afSi[0  , 0] := 1.00000E+01; afSi[0  , 1] := 6.81245E-01;
afSi[1  , 0] := 1.99800E+01; afSi[1  , 1] := 1.16318E-01;
afSi[2  , 0] := 2.99600E+01; afSi[2  , 1] := 1.82962E-01;
afSi[3  , 0] := 3.99400E+01; afSi[3  , 1] := 2.59571E-01;
afSi[4  , 0] := 4.99200E+01; afSi[4  , 1] := 3.13998E-01;
afSi[5  , 0] := 5.99000E+01; afSi[5  , 1] := 3.46321E-01;
afSi[6  , 0] := 6.98800E+01; afSi[6  , 1] := 3.63846E-01;
afSi[7  , 0] := 7.98600E+01; afSi[7  , 1] := 3.72124E-01;
afSi[8  , 0] := 8.98400E+01; afSi[8  , 1] := 3.76682E-01;
afSi[9  , 0] := 9.98200E+01; afSi[9  , 1] := 7.19156E+00;
afSi[10 , 0] := 1.09800E+02; afSi[10 , 1] := 8.20881E+00;
afSi[11 , 0] := 1.19780E+02; afSi[11 , 1] := 8.98291E+00;
afSi[12 , 0] := 1.29760E+02; afSi[12 , 1] := 9.38953E+00;
afSi[13 , 0] := 1.39740E+02; afSi[13 , 1] := 9.52436E+00;
afSi[14 , 0] := 1.49720E+02; afSi[14 , 1] := 1.01493E+01;
afSi[15 , 0] := 1.59700E+02; afSi[15 , 1] := 1.02033E+01;
afSi[16 , 0] := 1.69680E+02; afSi[16 , 1] := 9.94800E+00;
afSi[17 , 0] := 1.79660E+02; afSi[17 , 1] := 9.62733E+00;
afSi[18 , 0] := 1.89640E+02; afSi[18 , 1] := 9.27233E+00;
afSi[19 , 0] := 1.99620E+02; afSi[19 , 1] := 8.90204E+00;
afSi[20 , 0] := 2.09600E+02; afSi[20 , 1] := 8.52928E+00;
afSi[21 , 0] := 2.19580E+02; afSi[21 , 1] := 8.16149E+00;
afSi[22 , 0] := 2.29560E+02; afSi[22 , 1] := 7.80410E+00;
afSi[23 , 0] := 2.39540E+02; afSi[23 , 1] := 7.46085E+00;
afSi[24 , 0] := 2.49520E+02; afSi[24 , 1] := 7.13329E+00;
afSi[25 , 0] := 2.59500E+02; afSi[25 , 1] := 6.82216E+00;
afSi[26 , 0] := 2.69480E+02; afSi[26 , 1] := 6.52768E+00;
afSi[27 , 0] := 2.79460E+02; afSi[27 , 1] := 6.24948E+00;
afSi[28 , 0] := 2.89440E+02; afSi[28 , 1] := 5.98692E+00;
afSi[29 , 0] := 2.99420E+02; afSi[29 , 1] := 5.73954E+00;
afSi[30 , 0] := 3.09400E+02; afSi[30 , 1] := 5.50624E+00;
afSi[31 , 0] := 3.19380E+02; afSi[31 , 1] := 5.28643E+00;
afSi[32 , 0] := 3.29360E+02; afSi[32 , 1] := 5.07925E+00;
afSi[33 , 0] := 3.39340E+02; afSi[33 , 1] := 4.88381E+00;
afSi[34 , 0] := 3.49320E+02; afSi[34 , 1] := 4.69939E+00;
afSi[35 , 0] := 3.59300E+02; afSi[35 , 1] := 4.52528E+00;
afSi[36 , 0] := 3.69280E+02; afSi[36 , 1] := 4.36069E+00;
afSi[37 , 0] := 3.79260E+02; afSi[37 , 1] := 4.20508E+00;
afSi[38 , 0] := 3.89240E+02; afSi[38 , 1] := 4.05782E+00;
afSi[39 , 0] := 3.99220E+02; afSi[39 , 1] := 3.91835E+00;
afSi[40 , 0] := 4.09200E+02; afSi[40 , 1] := 3.78586E+00;
afSi[41 , 0] := 4.19180E+02; afSi[41 , 1] := 3.65995E+00;
afSi[42 , 0] := 4.29160E+02; afSi[42 , 1] := 3.54031E+00;
afSi[43 , 0] := 4.39140E+02; afSi[43 , 1] := 3.42645E+00;
afSi[44 , 0] := 4.49120E+02; afSi[44 , 1] := 3.31800E+00;
afSi[45 , 0] := 4.59100E+02; afSi[45 , 1] := 3.21480E+00;
afSi[46 , 0] := 4.69080E+02; afSi[46 , 1] := 3.11633E+00;
afSi[47 , 0] := 4.79060E+02; afSi[47 , 1] := 3.02250E+00;
afSi[48 , 0] := 4.89040E+02; afSi[48 , 1] := 2.93291E+00;
afSi[49 , 0] := 4.99020E+02; afSi[49 , 1] := 2.84732E+00;
afSi[50 , 0] := 5.09000E+02; afSi[50 , 1] := 2.76553E+00;
afSi[51 , 0] := 5.18980E+02; afSi[51 , 1] := 2.68738E+00;
afSi[52 , 0] := 5.28960E+02; afSi[52 , 1] := 2.61260E+00;
afSi[53 , 0] := 5.38940E+02; afSi[53 , 1] := 2.54091E+00;
afSi[54 , 0] := 5.48920E+02; afSi[54 , 1] := 2.47233E+00;
afSi[55 , 0] := 5.58900E+02; afSi[55 , 1] := 2.40663E+00;
afSi[56 , 0] := 5.68880E+02; afSi[56 , 1] := 2.34354E+00;
afSi[57 , 0] := 5.78860E+02; afSi[57 , 1] := 2.28303E+00;
afSi[58 , 0] := 5.88840E+02; afSi[58 , 1] := 2.22501E+00;
afSi[59 , 0] := 5.98820E+02; afSi[59 , 1] := 2.16915E+00;
afSi[60 , 0] := 6.08800E+02; afSi[60 , 1] := 2.11548E+00;
afSi[61 , 0] := 6.18780E+02; afSi[61 , 1] := 2.06389E+00;
afSi[62 , 0] := 6.28760E+02; afSi[62 , 1] := 2.01423E+00;
afSi[63 , 0] := 6.38740E+02; afSi[63 , 1] := 1.96636E+00;
afSi[64 , 0] := 6.48720E+02; afSi[64 , 1] := 1.92028E+00;
afSi[65 , 0] := 6.58700E+02; afSi[65 , 1] := 1.87584E+00;
afSi[66 , 0] := 6.68680E+02; afSi[66 , 1] := 1.83301E+00;
afSi[67 , 0] := 6.78660E+02; afSi[67 , 1] := 1.79173E+00;
afSi[68 , 0] := 6.88640E+02; afSi[68 , 1] := 1.75183E+00;
afSi[69 , 0] := 6.98620E+02; afSi[69 , 1] := 1.71334E+00;
afSi[70 , 0] := 7.08600E+02; afSi[70 , 1] := 1.67622E+00;
afSi[71 , 0] := 7.18580E+02; afSi[71 , 1] := 1.64031E+00;
afSi[72 , 0] := 7.28560E+02; afSi[72 , 1] := 1.60563E+00;
afSi[73 , 0] := 7.38540E+02; afSi[73 , 1] := 1.57210E+00;
afSi[74 , 0] := 7.48520E+02; afSi[74 , 1] := 1.53968E+00;
afSi[75 , 0] := 7.58500E+02; afSi[75 , 1] := 1.50829E+00;
afSi[76 , 0] := 7.68480E+02; afSi[76 , 1] := 1.47792E+00;
afSi[77 , 0] := 7.78460E+02; afSi[77 , 1] := 1.44845E+00;
afSi[78 , 0] := 7.88440E+02; afSi[78 , 1] := 1.41998E+00;
afSi[79 , 0] := 7.98420E+02; afSi[79 , 1] := 1.39240E+00;
afSi[80 , 0] := 8.08400E+02; afSi[80 , 1] := 1.36571E+00;
afSi[81 , 0] := 8.18380E+02; afSi[81 , 1] := 1.33980E+00;
afSi[82 , 0] := 8.28360E+02; afSi[82 , 1] := 1.31466E+00;
afSi[83 , 0] := 8.38340E+02; afSi[83 , 1] := 1.29025E+00;
afSi[84 , 0] := 8.48320E+02; afSi[84 , 1] := 1.26656E+00;
afSi[85 , 0] := 8.58300E+02; afSi[85 , 1] := 1.24365E+00;
afSi[86 , 0] := 8.68280E+02; afSi[86 , 1] := 1.22133E+00;
afSi[87 , 0] := 8.78260E+02; afSi[87 , 1] := 1.19966E+00;
afSi[88 , 0] := 8.88240E+02; afSi[88 , 1] := 1.17863E+00;
afSi[89 , 0] := 8.98220E+02; afSi[89 , 1] := 1.15820E+00;
afSi[90 , 0] := 9.08200E+02; afSi[90 , 1] := 1.13838E+00;
afSi[91 , 0] := 9.18180E+02; afSi[91 , 1] := 1.11907E+00;
afSi[92 , 0] := 9.28160E+02; afSi[92 , 1] := 1.10028E+00;
afSi[93 , 0] := 9.38140E+02; afSi[93 , 1] := 1.08204E+00;
afSi[94 , 0] := 9.48120E+02; afSi[94 , 1] := 1.06425E+00;
afSi[95 , 0] := 9.58100E+02; afSi[95 , 1] := 1.04696E+00;
afSi[96 , 0] := 9.68080E+02; afSi[96 , 1] := 1.03008E+00;
afSi[97 , 0] := 9.78060E+02; afSi[97 , 1] := 1.01368E+00;
afSi[98 , 0] := 9.88040E+02; afSi[98 , 1] := 9.97755E-01;
afSi[99 , 0] := 9.98020E+02; afSi[99 , 1] := 9.82162E-01;
afSi[100, 0] := 1.00800E+03; afSi[100, 1] := 9.65278E-01;
afSi[101, 0] := 1.01798E+03; afSi[101, 1] := 9.48403E-01;
afSi[102, 0] := 1.02796E+03; afSi[102, 1] := 9.32011E-01;
afSi[103, 0] := 1.03794E+03; afSi[103, 1] := 9.16062E-01;
afSi[104, 0] := 1.04792E+03; afSi[104, 1] := 9.00554E-01;
afSi[105, 0] := 1.05790E+03; afSi[105, 1] := 8.85466E-01;
afSi[106, 0] := 1.06788E+03; afSi[106, 1] := 8.70790E-01;
afSi[107, 0] := 1.07786E+03; afSi[107, 1] := 8.56506E-01;
afSi[108, 0] := 1.08784E+03; afSi[108, 1] := 8.42603E-01;
afSi[109, 0] := 1.09782E+03; afSi[109, 1] := 8.29061E-01;
afSi[110, 0] := 1.10780E+03; afSi[110, 1] := 8.15865E-01;
afSi[111, 0] := 1.11778E+03; afSi[111, 1] := 8.03013E-01;
afSi[112, 0] := 1.12776E+03; afSi[112, 1] := 7.90489E-01;
afSi[113, 0] := 1.13774E+03; afSi[113, 1] := 7.78275E-01;
afSi[114, 0] := 1.14772E+03; afSi[114, 1] := 7.66367E-01;
afSi[115, 0] := 1.15770E+03; afSi[115, 1] := 7.54761E-01;
afSi[116, 0] := 1.16768E+03; afSi[116, 1] := 7.43435E-01;
afSi[117, 0] := 1.17766E+03; afSi[117, 1] := 7.32388E-01;
afSi[118, 0] := 1.18764E+03; afSi[118, 1] := 7.21604E-01;
afSi[119, 0] := 1.19762E+03; afSi[119, 1] := 7.11077E-01;
afSi[120, 0] := 1.20760E+03; afSi[120, 1] := 7.00801E-01;
afSi[121, 0] := 1.21758E+03; afSi[121, 1] := 6.90760E-01;
afSi[122, 0] := 1.22756E+03; afSi[122, 1] := 6.80959E-01;
afSi[123, 0] := 1.23754E+03; afSi[123, 1] := 6.71384E-01;
afSi[124, 0] := 1.24752E+03; afSi[124, 1] := 6.62024E-01;
afSi[125, 0] := 1.25750E+03; afSi[125, 1] := 6.52877E-01;
afSi[126, 0] := 1.26748E+03; afSi[126, 1] := 6.43939E-01;
afSi[127, 0] := 1.27746E+03; afSi[127, 1] := 6.35196E-01;
afSi[128, 0] := 1.28744E+03; afSi[128, 1] := 6.26651E-01;
afSi[129, 0] := 1.29742E+03; afSi[129, 1] := 6.18294E-01;
afSi[130, 0] := 1.30740E+03; afSi[130, 1] := 6.10118E-01;
afSi[131, 0] := 1.31738E+03; afSi[131, 1] := 6.02115E-01;
afSi[132, 0] := 1.32736E+03; afSi[132, 1] := 5.94283E-01;
afSi[133, 0] := 1.33734E+03; afSi[133, 1] := 5.86618E-01;
afSi[134, 0] := 1.34732E+03; afSi[134, 1] := 5.79115E-01;
afSi[135, 0] := 1.35730E+03; afSi[135, 1] := 5.71772E-01;
afSi[136, 0] := 1.36728E+03; afSi[136, 1] := 5.64968E-01;
afSi[137, 0] := 1.37726E+03; afSi[137, 1] := 5.58124E-01;
afSi[138, 0] := 1.38724E+03; afSi[138, 1] := 5.51234E-01;
afSi[139, 0] := 1.39722E+03; afSi[139, 1] := 5.44489E-01;
afSi[140, 0] := 1.40720E+03; afSi[140, 1] := 5.37874E-01;
afSi[141, 0] := 1.41718E+03; afSi[141, 1] := 5.31392E-01;
afSi[142, 0] := 1.42716E+03; afSi[142, 1] := 5.25043E-01;
afSi[143, 0] := 1.43714E+03; afSi[143, 1] := 5.18819E-01;
afSi[144, 0] := 1.44712E+03; afSi[144, 1] := 5.12719E-01;
afSi[145, 0] := 1.45710E+03; afSi[145, 1] := 5.06739E-01;
afSi[146, 0] := 1.46708E+03; afSi[146, 1] := 5.00878E-01;
afSi[147, 0] := 1.47706E+03; afSi[147, 1] := 4.95126E-01;
afSi[148, 0] := 1.48704E+03; afSi[148, 1] := 4.89482E-01;
afSi[149, 0] := 1.49702E+03; afSi[149, 1] := 4.83950E-01;
afSi[150, 0] := 1.50700E+03; afSi[150, 1] := 4.78523E-01;
afSi[151, 0] := 1.51698E+03; afSi[151, 1] := 4.73196E-01;
afSi[152, 0] := 1.52696E+03; afSi[152, 1] := 4.67971E-01;
afSi[153, 0] := 1.53694E+03; afSi[153, 1] := 4.62844E-01;
afSi[154, 0] := 1.54692E+03; afSi[154, 1] := 4.57811E-01;
afSi[155, 0] := 1.55690E+03; afSi[155, 1] := 4.52871E-01;
afSi[156, 0] := 1.56688E+03; afSi[156, 1] := 4.48024E-01;
afSi[157, 0] := 1.57686E+03; afSi[157, 1] := 4.43265E-01;
afSi[158, 0] := 1.58684E+03; afSi[158, 1] := 4.38596E-01;
afSi[159, 0] := 1.59682E+03; afSi[159, 1] := 4.34013E-01;
afSi[160, 0] := 1.60680E+03; afSi[160, 1] := 4.29517E-01;
afSi[161, 0] := 1.61678E+03; afSi[161, 1] := 4.25105E-01;
afSi[162, 0] := 1.62676E+03; afSi[162, 1] := 4.20771E-01;
afSi[163, 0] := 1.63674E+03; afSi[163, 1] := 4.16519E-01;
afSi[164, 0] := 1.64672E+03; afSi[164, 1] := 4.12348E-01;
afSi[165, 0] := 1.65670E+03; afSi[165, 1] := 4.08254E-01;
afSi[166, 0] := 1.66668E+03; afSi[166, 1] := 4.04241E-01;
afSi[167, 0] := 1.67666E+03; afSi[167, 1] := 4.00302E-01;
afSi[168, 0] := 1.68664E+03; afSi[168, 1] := 3.96446E-01;
afSi[169, 0] := 1.69662E+03; afSi[169, 1] := 3.92678E-01;
afSi[170, 0] := 1.70660E+03; afSi[170, 1] := 3.88985E-01;
afSi[171, 0] := 1.71658E+03; afSi[171, 1] := 3.85390E-01;
afSi[172, 0] := 1.72656E+03; afSi[172, 1] := 3.81869E-01;
afSi[173, 0] := 1.73654E+03; afSi[173, 1] := 3.78464E-01;
afSi[174, 0] := 1.74652E+03; afSi[174, 1] := 3.75164E-01;
afSi[175, 0] := 1.75650E+03; afSi[175, 1] := 3.71977E-01;
afSi[176, 0] := 1.76648E+03; afSi[176, 1] := 3.68994E-01;
afSi[177, 0] := 1.77646E+03; afSi[177, 1] := 3.66114E-01;
afSi[178, 0] := 1.78644E+03; afSi[178, 1] := 3.63726E-01;
afSi[179, 0] := 1.79642E+03; afSi[179, 1] := 3.61633E-01;
afSi[180, 0] := 1.80640E+03; afSi[180, 1] := 3.60725E-01;
afSi[181, 0] := 1.81638E+03; afSi[181, 1] := 3.61625E-01;
afSi[182, 0] := 1.82636E+03; afSi[182, 1] := 3.68918E-01;
afSi[183, 0] := 1.83634E+03; afSi[183, 1] := 4.60263E-01;
afSi[184, 0] := 1.84632E+03; afSi[184, 1] := 4.04826E+00;
afSi[185, 0] := 1.85630E+03; afSi[185, 1] := 4.04956E+00;
afSi[186, 0] := 1.86628E+03; afSi[186, 1] := 4.03746E+00;
afSi[187, 0] := 1.87626E+03; afSi[187, 1] := 4.02159E+00;
afSi[188, 0] := 1.88624E+03; afSi[188, 1] := 4.00531E+00;
afSi[189, 0] := 1.89622E+03; afSi[189, 1] := 3.98804E+00;
afSi[190, 0] := 1.90620E+03; afSi[190, 1] := 3.97090E+00;
afSi[191, 0] := 1.91618E+03; afSi[191, 1] := 3.95361E+00;
afSi[192, 0] := 1.92616E+03; afSi[192, 1] := 3.93518E+00;
afSi[193, 0] := 1.93614E+03; afSi[193, 1] := 3.91177E+00;
afSi[194, 0] := 1.94612E+03; afSi[194, 1] := 3.88771E+00;
afSi[195, 0] := 1.95610E+03; afSi[195, 1] := 3.86151E+00;
afSi[196, 0] := 1.96608E+03; afSi[196, 1] := 3.83528E+00;
afSi[197, 0] := 1.97606E+03; afSi[197, 1] := 3.80869E+00;
afSi[198, 0] := 1.98604E+03; afSi[198, 1] := 3.78211E+00;
afSi[199, 0] := 1.99602E+03; afSi[199, 1] := 3.75528E+00;
afSi[200, 0] := 2.00600E+03; afSi[200, 1] := 3.72847E+00;
afSi[201, 0] := 2.01598E+03; afSi[201, 1] := 3.70146E+00;
afSi[202, 0] := 2.02596E+03; afSi[202, 1] := 3.67455E+00;
afSi[203, 0] := 2.03594E+03; afSi[203, 1] := 3.64755E+00;
afSi[204, 0] := 2.04592E+03; afSi[204, 1] := 3.62067E+00;
afSi[205, 0] := 2.05590E+03; afSi[205, 1] := 3.59369E+00;
afSi[206, 0] := 2.06588E+03; afSi[206, 1] := 3.56688E+00;
afSi[207, 0] := 2.07586E+03; afSi[207, 1] := 3.54005E+00;
afSi[208, 0] := 2.08584E+03; afSi[208, 1] := 3.51346E+00;
afSi[209, 0] := 2.09582E+03; afSi[209, 1] := 3.48686E+00;
afSi[210, 0] := 2.10580E+03; afSi[210, 1] := 3.46054E+00;
afSi[211, 0] := 2.11578E+03; afSi[211, 1] := 3.43418E+00;
afSi[212, 0] := 2.12576E+03; afSi[212, 1] := 3.40813E+00;
afSi[213, 0] := 2.13574E+03; afSi[213, 1] := 3.38209E+00;
afSi[214, 0] := 2.14572E+03; afSi[214, 1] := 3.35637E+00;
afSi[215, 0] := 2.15570E+03; afSi[215, 1] := 3.33075E+00;
afSi[216, 0] := 2.16568E+03; afSi[216, 1] := 3.30542E+00;
afSi[217, 0] := 2.17566E+03; afSi[217, 1] := 3.28023E+00;
afSi[218, 0] := 2.18564E+03; afSi[218, 1] := 3.25529E+00;
afSi[219, 0] := 2.19562E+03; afSi[219, 1] := 3.23054E+00;
afSi[220, 0] := 2.20560E+03; afSi[220, 1] := 3.20602E+00;
afSi[221, 0] := 2.21558E+03; afSi[221, 1] := 3.18174E+00;
afSi[222, 0] := 2.22556E+03; afSi[222, 1] := 3.15767E+00;
afSi[223, 0] := 2.23554E+03; afSi[223, 1] := 3.13387E+00;
afSi[224, 0] := 2.24552E+03; afSi[224, 1] := 3.11029E+00;
afSi[225, 0] := 2.25550E+03; afSi[225, 1] := 3.08699E+00;
afSi[226, 0] := 2.26548E+03; afSi[226, 1] := 3.06393E+00;
afSi[227, 0] := 2.27546E+03; afSi[227, 1] := 3.04114E+00;
afSi[228, 0] := 2.28544E+03; afSi[228, 1] := 3.01857E+00;
afSi[229, 0] := 2.29542E+03; afSi[229, 1] := 2.99625E+00;
afSi[230, 0] := 2.30540E+03; afSi[230, 1] := 2.97429E+00;
afSi[231, 0] := 2.31538E+03; afSi[231, 1] := 2.95276E+00;
afSi[232, 0] := 2.32536E+03; afSi[232, 1] := 2.93145E+00;
afSi[233, 0] := 2.33534E+03; afSi[233, 1] := 2.91014E+00;
afSi[234, 0] := 2.34532E+03; afSi[234, 1] := 2.88908E+00;
afSi[235, 0] := 2.35530E+03; afSi[235, 1] := 2.86831E+00;
afSi[236, 0] := 2.36528E+03; afSi[236, 1] := 2.84780E+00;
afSi[237, 0] := 2.37526E+03; afSi[237, 1] := 2.82758E+00;
afSi[238, 0] := 2.38524E+03; afSi[238, 1] := 2.80769E+00;
afSi[239, 0] := 2.39522E+03; afSi[239, 1] := 2.78804E+00;
afSi[240, 0] := 2.40520E+03; afSi[240, 1] := 2.76923E+00;
afSi[241, 0] := 2.41518E+03; afSi[241, 1] := 2.75063E+00;
afSi[242, 0] := 2.42516E+03; afSi[242, 1] := 2.73228E+00;
afSi[243, 0] := 2.43514E+03; afSi[243, 1] := 2.71415E+00;
afSi[244, 0] := 2.44512E+03; afSi[244, 1] := 2.69621E+00;
afSi[245, 0] := 2.45510E+03; afSi[245, 1] := 2.67847E+00;
afSi[246, 0] := 2.46508E+03; afSi[246, 1] := 2.66091E+00;
afSi[247, 0] := 2.47506E+03; afSi[247, 1] := 2.64357E+00;
afSi[248, 0] := 2.48504E+03; afSi[248, 1] := 2.62642E+00;
afSi[249, 0] := 2.49502E+03; afSi[249, 1] := 2.60947E+00;
afSi[250, 0] := 2.50500E+03; afSi[250, 1] := 2.59273E+00;
afSi[251, 0] := 2.51498E+03; afSi[251, 1] := 2.57616E+00;
afSi[252, 0] := 2.52496E+03; afSi[252, 1] := 2.55981E+00;
afSi[253, 0] := 2.53494E+03; afSi[253, 1] := 2.54364E+00;
afSi[254, 0] := 2.54492E+03; afSi[254, 1] := 2.52764E+00;
afSi[255, 0] := 2.55490E+03; afSi[255, 1] := 2.51181E+00;
afSi[256, 0] := 2.56488E+03; afSi[256, 1] := 2.49615E+00;
afSi[257, 0] := 2.57486E+03; afSi[257, 1] := 2.48063E+00;
afSi[258, 0] := 2.58484E+03; afSi[258, 1] := 2.46527E+00;
afSi[259, 0] := 2.59482E+03; afSi[259, 1] := 2.45007E+00;
afSi[260, 0] := 2.60480E+03; afSi[260, 1] := 2.43508E+00;
afSi[261, 0] := 2.61478E+03; afSi[261, 1] := 2.42024E+00;
afSi[262, 0] := 2.62476E+03; afSi[262, 1] := 2.40554E+00;
afSi[263, 0] := 2.63474E+03; afSi[263, 1] := 2.39098E+00;
afSi[264, 0] := 2.64472E+03; afSi[264, 1] := 2.37657E+00;
afSi[265, 0] := 2.65470E+03; afSi[265, 1] := 2.36233E+00;
afSi[266, 0] := 2.66468E+03; afSi[266, 1] := 2.34824E+00;
afSi[267, 0] := 2.67466E+03; afSi[267, 1] := 2.33428E+00;
afSi[268, 0] := 2.68464E+03; afSi[268, 1] := 2.32046E+00;
afSi[269, 0] := 2.69462E+03; afSi[269, 1] := 2.30677E+00;
afSi[270, 0] := 2.70460E+03; afSi[270, 1] := 2.29321E+00;
afSi[271, 0] := 2.71458E+03; afSi[271, 1] := 2.27979E+00;
afSi[272, 0] := 2.72456E+03; afSi[272, 1] := 2.26650E+00;
afSi[273, 0] := 2.73454E+03; afSi[273, 1] := 2.25334E+00;
afSi[274, 0] := 2.74452E+03; afSi[274, 1] := 2.24031E+00;
afSi[275, 0] := 2.75450E+03; afSi[275, 1] := 2.22740E+00;
afSi[276, 0] := 2.76448E+03; afSi[276, 1] := 2.21459E+00;
afSi[277, 0] := 2.77446E+03; afSi[277, 1] := 2.20189E+00;
afSi[278, 0] := 2.78444E+03; afSi[278, 1] := 2.18931E+00;
afSi[279, 0] := 2.79442E+03; afSi[279, 1] := 2.17684E+00;
afSi[280, 0] := 2.80440E+03; afSi[280, 1] := 2.16448E+00;
afSi[281, 0] := 2.81438E+03; afSi[281, 1] := 2.15222E+00;
afSi[282, 0] := 2.82436E+03; afSi[282, 1] := 2.14007E+00;
afSi[283, 0] := 2.83434E+03; afSi[283, 1] := 2.12803E+00;
afSi[284, 0] := 2.84432E+03; afSi[284, 1] := 2.11606E+00;
afSi[285, 0] := 2.85430E+03; afSi[285, 1] := 2.10418E+00;
afSi[286, 0] := 2.86428E+03; afSi[286, 1] := 2.09242E+00;
afSi[287, 0] := 2.87426E+03; afSi[287, 1] := 2.08079E+00;
afSi[288, 0] := 2.88424E+03; afSi[288, 1] := 2.06926E+00;
afSi[289, 0] := 2.89422E+03; afSi[289, 1] := 2.05783E+00;
afSi[290, 0] := 2.90420E+03; afSi[290, 1] := 2.04650E+00;
afSi[291, 0] := 2.91418E+03; afSi[291, 1] := 2.03527E+00;
afSi[292, 0] := 2.92416E+03; afSi[292, 1] := 2.02413E+00;
afSi[293, 0] := 2.93414E+03; afSi[293, 1] := 2.01310E+00;
afSi[294, 0] := 2.94412E+03; afSi[294, 1] := 2.00215E+00;
afSi[295, 0] := 2.95410E+03; afSi[295, 1] := 1.99131E+00;
afSi[296, 0] := 2.96408E+03; afSi[296, 1] := 1.98056E+00;
afSi[297, 0] := 2.97406E+03; afSi[297, 1] := 1.96990E+00;
afSi[298, 0] := 2.98404E+03; afSi[298, 1] := 1.95926E+00;
afSi[299, 0] := 2.99402E+03; afSi[299, 1] := 1.94855E+00;
afSi[300, 0] := 3.00400E+03; afSi[300, 1] := 1.93793E+00;
afSi[301, 0] := 3.01398E+03; afSi[301, 1] := 1.92730E+00;
afSi[302, 0] := 3.02396E+03; afSi[302, 1] := 1.91653E+00;
afSi[303, 0] := 3.03394E+03; afSi[303, 1] := 1.90585E+00;
afSi[304, 0] := 3.04392E+03; afSi[304, 1] := 1.89527E+00;
afSi[305, 0] := 3.05390E+03; afSi[305, 1] := 1.88476E+00;
afSi[306, 0] := 3.06388E+03; afSi[306, 1] := 1.87435E+00;
afSi[307, 0] := 3.07386E+03; afSi[307, 1] := 1.86404E+00;
afSi[308, 0] := 3.08384E+03; afSi[308, 1] := 1.85383E+00;
afSi[309, 0] := 3.09382E+03; afSi[309, 1] := 1.84371E+00;
afSi[310, 0] := 3.10380E+03; afSi[310, 1] := 1.83367E+00;
afSi[311, 0] := 3.11378E+03; afSi[311, 1] := 1.82372E+00;
afSi[312, 0] := 3.12376E+03; afSi[312, 1] := 1.81385E+00;
afSi[313, 0] := 3.13374E+03; afSi[313, 1] := 1.80407E+00;
afSi[314, 0] := 3.14372E+03; afSi[314, 1] := 1.79437E+00;
afSi[315, 0] := 3.15370E+03; afSi[315, 1] := 1.78475E+00;
afSi[316, 0] := 3.16368E+03; afSi[316, 1] := 1.77521E+00;
afSi[317, 0] := 3.17366E+03; afSi[317, 1] := 1.76575E+00;
afSi[318, 0] := 3.18364E+03; afSi[318, 1] := 1.75637E+00;
afSi[319, 0] := 3.19362E+03; afSi[319, 1] := 1.74707E+00;
afSi[320, 0] := 3.20360E+03; afSi[320, 1] := 1.73785E+00;
afSi[321, 0] := 3.21358E+03; afSi[321, 1] := 1.72870E+00;
afSi[322, 0] := 3.22356E+03; afSi[322, 1] := 1.71964E+00;
afSi[323, 0] := 3.23354E+03; afSi[323, 1] := 1.71064E+00;
afSi[324, 0] := 3.24352E+03; afSi[324, 1] := 1.70173E+00;
afSi[325, 0] := 3.25350E+03; afSi[325, 1] := 1.69289E+00;
afSi[326, 0] := 3.26348E+03; afSi[326, 1] := 1.68412E+00;
afSi[327, 0] := 3.27346E+03; afSi[327, 1] := 1.67543E+00;
afSi[328, 0] := 3.28344E+03; afSi[328, 1] := 1.66681E+00;
afSi[329, 0] := 3.29342E+03; afSi[329, 1] := 1.65826E+00;
afSi[330, 0] := 3.30340E+03; afSi[330, 1] := 1.64979E+00;
afSi[331, 0] := 3.31338E+03; afSi[331, 1] := 1.64139E+00;
afSi[332, 0] := 3.32336E+03; afSi[332, 1] := 1.63306E+00;
afSi[333, 0] := 3.33334E+03; afSi[333, 1] := 1.62477E+00;
afSi[334, 0] := 3.34332E+03; afSi[334, 1] := 1.61655E+00;
afSi[335, 0] := 3.35330E+03; afSi[335, 1] := 1.60840E+00;
afSi[336, 0] := 3.36328E+03; afSi[336, 1] := 1.60032E+00;
afSi[337, 0] := 3.37326E+03; afSi[337, 1] := 1.59231E+00;
afSi[338, 0] := 3.38324E+03; afSi[338, 1] := 1.58436E+00;
afSi[339, 0] := 3.39322E+03; afSi[339, 1] := 1.57647E+00;
afSi[340, 0] := 3.40320E+03; afSi[340, 1] := 1.56864E+00;
afSi[341, 0] := 3.41318E+03; afSi[341, 1] := 1.56086E+00;
afSi[342, 0] := 3.42316E+03; afSi[342, 1] := 1.55315E+00;
afSi[343, 0] := 3.43314E+03; afSi[343, 1] := 1.54551E+00;
afSi[344, 0] := 3.44312E+03; afSi[344, 1] := 1.53793E+00;
afSi[345, 0] := 3.45310E+03; afSi[345, 1] := 1.53041E+00;
afSi[346, 0] := 3.46308E+03; afSi[346, 1] := 1.52295E+00;
afSi[347, 0] := 3.47306E+03; afSi[347, 1] := 1.51554E+00;
afSi[348, 0] := 3.48304E+03; afSi[348, 1] := 1.50818E+00;
afSi[349, 0] := 3.49302E+03; afSi[349, 1] := 1.50089E+00;
afSi[350, 0] := 3.50300E+03; afSi[350, 1] := 1.49366E+00;
afSi[351, 0] := 3.51298E+03; afSi[351, 1] := 1.48649E+00;
afSi[352, 0] := 3.52296E+03; afSi[352, 1] := 1.47938E+00;
afSi[353, 0] := 3.53294E+03; afSi[353, 1] := 1.47232E+00;
afSi[354, 0] := 3.54292E+03; afSi[354, 1] := 1.46528E+00;
afSi[355, 0] := 3.55290E+03; afSi[355, 1] := 1.45830E+00;
afSi[356, 0] := 3.56288E+03; afSi[356, 1] := 1.45137E+00;
afSi[357, 0] := 3.57286E+03; afSi[357, 1] := 1.44451E+00;
afSi[358, 0] := 3.58284E+03; afSi[358, 1] := 1.43770E+00;
afSi[359, 0] := 3.59282E+03; afSi[359, 1] := 1.43095E+00;
afSi[360, 0] := 3.60280E+03; afSi[360, 1] := 1.42425E+00;
afSi[361, 0] := 3.61278E+03; afSi[361, 1] := 1.41760E+00;
afSi[362, 0] := 3.62276E+03; afSi[362, 1] := 1.41099E+00;
afSi[363, 0] := 3.63274E+03; afSi[363, 1] := 1.40444E+00;
afSi[364, 0] := 3.64272E+03; afSi[364, 1] := 1.39793E+00;
afSi[365, 0] := 3.65270E+03; afSi[365, 1] := 1.39148E+00;
afSi[366, 0] := 3.66268E+03; afSi[366, 1] := 1.38507E+00;
afSi[367, 0] := 3.67266E+03; afSi[367, 1] := 1.37870E+00;
afSi[368, 0] := 3.68264E+03; afSi[368, 1] := 1.37200E+00;
afSi[369, 0] := 3.69262E+03; afSi[369, 1] := 1.36529E+00;
afSi[370, 0] := 3.70260E+03; afSi[370, 1] := 1.35864E+00;
afSi[371, 0] := 3.71258E+03; afSi[371, 1] := 1.35202E+00;
afSi[372, 0] := 3.72256E+03; afSi[372, 1] := 1.34540E+00;
afSi[373, 0] := 3.73254E+03; afSi[373, 1] := 1.33883E+00;
afSi[374, 0] := 3.74252E+03; afSi[374, 1] := 1.33231E+00;
afSi[375, 0] := 3.75250E+03; afSi[375, 1] := 1.32585E+00;
afSi[376, 0] := 3.76248E+03; afSi[376, 1] := 1.31944E+00;
afSi[377, 0] := 3.77246E+03; afSi[377, 1] := 1.31308E+00;
afSi[378, 0] := 3.78244E+03; afSi[378, 1] := 1.30677E+00;
afSi[379, 0] := 3.79242E+03; afSi[379, 1] := 1.30050E+00;
afSi[380, 0] := 3.80240E+03; afSi[380, 1] := 1.29427E+00;
afSi[381, 0] := 3.81238E+03; afSi[381, 1] := 1.28809E+00;
afSi[382, 0] := 3.82236E+03; afSi[382, 1] := 1.28195E+00;
afSi[383, 0] := 3.83234E+03; afSi[383, 1] := 1.27586E+00;
afSi[384, 0] := 3.84232E+03; afSi[384, 1] := 1.26980E+00;
afSi[385, 0] := 3.85230E+03; afSi[385, 1] := 1.26380E+00;
afSi[386, 0] := 3.86228E+03; afSi[386, 1] := 1.25784E+00;
afSi[387, 0] := 3.87226E+03; afSi[387, 1] := 1.25194E+00;
afSi[388, 0] := 3.88224E+03; afSi[388, 1] := 1.24608E+00;
afSi[389, 0] := 3.89222E+03; afSi[389, 1] := 1.24027E+00;
afSi[390, 0] := 3.90220E+03; afSi[390, 1] := 1.23449E+00;
afSi[391, 0] := 3.91218E+03; afSi[391, 1] := 1.22873E+00;
afSi[392, 0] := 3.92216E+03; afSi[392, 1] := 1.22302E+00;
afSi[393, 0] := 3.93214E+03; afSi[393, 1] := 1.21734E+00;
afSi[394, 0] := 3.94212E+03; afSi[394, 1] := 1.21172E+00;
afSi[395, 0] := 3.95210E+03; afSi[395, 1] := 1.20615E+00;
afSi[396, 0] := 3.96208E+03; afSi[396, 1] := 1.20062E+00;
afSi[397, 0] := 3.97206E+03; afSi[397, 1] := 1.19513E+00;
afSi[398, 0] := 3.98204E+03; afSi[398, 1] := 1.18967E+00;
afSi[399, 0] := 3.99202E+03; afSi[399, 1] := 1.18423E+00;
afSi[400, 0] := 4.00200E+03; afSi[400, 1] := 1.17884E+00;
afSi[401, 0] := 4.01198E+03; afSi[401, 1] := 1.17348E+00;
afSi[402, 0] := 4.02196E+03; afSi[402, 1] := 1.16816E+00;
afSi[403, 0] := 4.03194E+03; afSi[403, 1] := 1.16291E+00;
afSi[404, 0] := 4.04192E+03; afSi[404, 1] := 1.15769E+00;
afSi[405, 0] := 4.05190E+03; afSi[405, 1] := 1.15250E+00;
afSi[406, 0] := 4.06188E+03; afSi[406, 1] := 1.14735E+00;
afSi[407, 0] := 4.07186E+03; afSi[407, 1] := 1.14222E+00;
afSi[408, 0] := 4.08184E+03; afSi[408, 1] := 1.13712E+00;
afSi[409, 0] := 4.09182E+03; afSi[409, 1] := 1.13206E+00;
afSi[410, 0] := 4.10180E+03; afSi[410, 1] := 1.12703E+00;
afSi[411, 0] := 4.11178E+03; afSi[411, 1] := 1.12205E+00;
afSi[412, 0] := 4.12176E+03; afSi[412, 1] := 1.11710E+00;
afSi[413, 0] := 4.13174E+03; afSi[413, 1] := 1.11218E+00;
afSi[414, 0] := 4.14172E+03; afSi[414, 1] := 1.10730E+00;
afSi[415, 0] := 4.15170E+03; afSi[415, 1] := 1.10246E+00;
afSi[416, 0] := 4.16168E+03; afSi[416, 1] := 1.09765E+00;
afSi[417, 0] := 4.17166E+03; afSi[417, 1] := 1.09287E+00;
afSi[418, 0] := 4.18164E+03; afSi[418, 1] := 1.08812E+00;
afSi[419, 0] := 4.19162E+03; afSi[419, 1] := 1.08340E+00;
afSi[420, 0] := 4.20160E+03; afSi[420, 1] := 1.07870E+00;
afSi[421, 0] := 4.21158E+03; afSi[421, 1] := 1.07404E+00;
afSi[422, 0] := 4.22156E+03; afSi[422, 1] := 1.06940E+00;
afSi[423, 0] := 4.23154E+03; afSi[423, 1] := 1.06481E+00;
afSi[424, 0] := 4.24152E+03; afSi[424, 1] := 1.06025E+00;
afSi[425, 0] := 4.25150E+03; afSi[425, 1] := 1.05572E+00;
afSi[426, 0] := 4.26148E+03; afSi[426, 1] := 1.05122E+00;
afSi[427, 0] := 4.27146E+03; afSi[427, 1] := 1.04674E+00;
afSi[428, 0] := 4.28144E+03; afSi[428, 1] := 1.04229E+00;
afSi[429, 0] := 4.29142E+03; afSi[429, 1] := 1.03787E+00;
afSi[430, 0] := 4.30140E+03; afSi[430, 1] := 1.03347E+00;
afSi[431, 0] := 4.31138E+03; afSi[431, 1] := 1.02911E+00;
afSi[432, 0] := 4.32136E+03; afSi[432, 1] := 1.02479E+00;
afSi[433, 0] := 4.33134E+03; afSi[433, 1] := 1.02050E+00;
afSi[434, 0] := 4.34132E+03; afSi[434, 1] := 1.01623E+00;
afSi[435, 0] := 4.35130E+03; afSi[435, 1] := 1.01199E+00;
afSi[436, 0] := 4.36128E+03; afSi[436, 1] := 1.00776E+00;
afSi[437, 0] := 4.37126E+03; afSi[437, 1] := 1.00356E+00;
afSi[438, 0] := 4.38124E+03; afSi[438, 1] := 9.99379E-01;
afSi[439, 0] := 4.39122E+03; afSi[439, 1] := 9.95230E-01;
afSi[440, 0] := 4.40120E+03; afSi[440, 1] := 9.91115E-01;
afSi[441, 0] := 4.41118E+03; afSi[441, 1] := 9.87029E-01;
afSi[442, 0] := 4.42116E+03; afSi[442, 1] := 9.82970E-01;
afSi[443, 0] := 4.43114E+03; afSi[443, 1] := 9.78937E-01;
afSi[444, 0] := 4.44112E+03; afSi[444, 1] := 9.74929E-01;
afSi[445, 0] := 4.45110E+03; afSi[445, 1] := 9.70947E-01;
afSi[446, 0] := 4.46108E+03; afSi[446, 1] := 9.66989E-01;
afSi[447, 0] := 4.47106E+03; afSi[447, 1] := 9.63057E-01;
afSi[448, 0] := 4.48104E+03; afSi[448, 1] := 9.59149E-01;
afSi[449, 0] := 4.49102E+03; afSi[449, 1] := 9.55265E-01;
afSi[450, 0] := 4.50100E+03; afSi[450, 1] := 9.51404E-01;
afSi[451, 0] := 4.51098E+03; afSi[451, 1] := 9.47568E-01;
afSi[452, 0] := 4.52096E+03; afSi[452, 1] := 9.43756E-01;
afSi[453, 0] := 4.53094E+03; afSi[453, 1] := 9.39968E-01;
afSi[454, 0] := 4.54092E+03; afSi[454, 1] := 9.36205E-01;
afSi[455, 0] := 4.55090E+03; afSi[455, 1] := 9.32465E-01;
afSi[456, 0] := 4.56088E+03; afSi[456, 1] := 9.28749E-01;
afSi[457, 0] := 4.57086E+03; afSi[457, 1] := 9.25055E-01;
afSi[458, 0] := 4.58084E+03; afSi[458, 1] := 9.21383E-01;
afSi[459, 0] := 4.59082E+03; afSi[459, 1] := 9.17734E-01;
afSi[460, 0] := 4.60080E+03; afSi[460, 1] := 9.14107E-01;
afSi[461, 0] := 4.61078E+03; afSi[461, 1] := 9.10502E-01;
afSi[462, 0] := 4.62076E+03; afSi[462, 1] := 9.06919E-01;
afSi[463, 0] := 4.63074E+03; afSi[463, 1] := 9.03358E-01;
afSi[464, 0] := 4.64072E+03; afSi[464, 1] := 8.99819E-01;
afSi[465, 0] := 4.65070E+03; afSi[465, 1] := 8.96301E-01;
afSi[466, 0] := 4.66068E+03; afSi[466, 1] := 8.92804E-01;
afSi[467, 0] := 4.67066E+03; afSi[467, 1] := 8.89329E-01;
afSi[468, 0] := 4.68064E+03; afSi[468, 1] := 8.85876E-01;
afSi[469, 0] := 4.69062E+03; afSi[469, 1] := 8.82444E-01;
afSi[470, 0] := 4.70060E+03; afSi[470, 1] := 8.79032E-01;
afSi[471, 0] := 4.71058E+03; afSi[471, 1] := 8.75640E-01;
afSi[472, 0] := 4.72056E+03; afSi[472, 1] := 8.72267E-01;
afSi[473, 0] := 4.73054E+03; afSi[473, 1] := 8.68914E-01;
afSi[474, 0] := 4.74052E+03; afSi[474, 1] := 8.65581E-01;
afSi[475, 0] := 4.75050E+03; afSi[475, 1] := 8.62268E-01;
afSi[476, 0] := 4.76048E+03; afSi[476, 1] := 8.58974E-01;
afSi[477, 0] := 4.77046E+03; afSi[477, 1] := 8.55702E-01;
afSi[478, 0] := 4.78044E+03; afSi[478, 1] := 8.52448E-01;
afSi[479, 0] := 4.79042E+03; afSi[479, 1] := 8.49214E-01;
afSi[480, 0] := 4.80040E+03; afSi[480, 1] := 8.45998E-01;
afSi[481, 0] := 4.81038E+03; afSi[481, 1] := 8.42802E-01;
afSi[482, 0] := 4.82036E+03; afSi[482, 1] := 8.39624E-01;
afSi[483, 0] := 4.83034E+03; afSi[483, 1] := 8.36465E-01;
afSi[484, 0] := 4.84032E+03; afSi[484, 1] := 8.33325E-01;
afSi[485, 0] := 4.85030E+03; afSi[485, 1] := 8.30202E-01;
afSi[486, 0] := 4.86028E+03; afSi[486, 1] := 8.27098E-01;
afSi[487, 0] := 4.87026E+03; afSi[487, 1] := 8.24011E-01;
afSi[488, 0] := 4.88024E+03; afSi[488, 1] := 8.20942E-01;
afSi[489, 0] := 4.89022E+03; afSi[489, 1] := 8.17890E-01;
afSi[490, 0] := 4.90020E+03; afSi[490, 1] := 8.14857E-01;
afSi[491, 0] := 4.91018E+03; afSi[491, 1] := 8.11840E-01;
afSi[492, 0] := 4.92016E+03; afSi[492, 1] := 8.08842E-01;
afSi[493, 0] := 4.93014E+03; afSi[493, 1] := 8.05860E-01;
afSi[494, 0] := 4.94012E+03; afSi[494, 1] := 8.02895E-01;
afSi[495, 0] := 4.95010E+03; afSi[495, 1] := 7.99947E-01;
afSi[496, 0] := 4.96008E+03; afSi[496, 1] := 7.97017E-01;
afSi[497, 0] := 4.97006E+03; afSi[497, 1] := 7.94104E-01;
afSi[498, 0] := 4.98004E+03; afSi[498, 1] := 7.91208E-01;
afSi[499, 0] := 4.99002E+03; afSi[499, 1] := 7.88327E-01;
afSi[500, 0] := 5.00000E+03; afSi[500, 1] := 7.85463E-01;
afSi[501, 0] := 5.05000E+03; afSi[501, 1] := 7.71346E-01;
afSi[502, 0] := 5.10000E+03; afSi[502, 1] := 7.57615E-01;
afSi[503, 0] := 5.15000E+03; afSi[503, 1] := 7.44268E-01;
afSi[504, 0] := 5.20000E+03; afSi[504, 1] := 7.31279E-01;
afSi[505, 0] := 5.25000E+03; afSi[505, 1] := 7.18637E-01;
afSi[506, 0] := 5.30000E+03; afSi[506, 1] := 7.06325E-01;
afSi[507, 0] := 5.35000E+03; afSi[507, 1] := 6.94343E-01;
afSi[508, 0] := 5.40000E+03; afSi[508, 1] := 6.82669E-01;
afSi[509, 0] := 5.45000E+03; afSi[509, 1] := 6.71298E-01;
afSi[510, 0] := 5.50000E+03; afSi[510, 1] := 6.60221E-01;
afSi[511, 0] := 5.55000E+03; afSi[511, 1] := 6.49422E-01;
afSi[512, 0] := 5.60000E+03; afSi[512, 1] := 6.38895E-01;
afSi[513, 0] := 5.65000E+03; afSi[513, 1] := 6.28633E-01;
afSi[514, 0] := 5.70000E+03; afSi[514, 1] := 6.18619E-01;
afSi[515, 0] := 5.75000E+03; afSi[515, 1] := 6.08855E-01;
afSi[516, 0] := 5.80000E+03; afSi[516, 1] := 5.99328E-01;
afSi[517, 0] := 5.85000E+03; afSi[517, 1] := 5.90032E-01;
afSi[518, 0] := 5.90000E+03; afSi[518, 1] := 5.80957E-01;
afSi[519, 0] := 5.95000E+03; afSi[519, 1] := 5.72095E-01;
afSi[520, 0] := 6.00000E+03; afSi[520, 1] := 5.63442E-01;
afSi[521, 0] := 6.05000E+03; afSi[521, 1] := 5.54992E-01;
afSi[522, 0] := 6.10000E+03; afSi[522, 1] := 5.46736E-01;
afSi[523, 0] := 6.15000E+03; afSi[523, 1] := 5.38668E-01;
afSi[524, 0] := 6.20000E+03; afSi[524, 1] := 5.30779E-01;
afSi[525, 0] := 6.25000E+03; afSi[525, 1] := 5.23070E-01;
afSi[526, 0] := 6.30000E+03; afSi[526, 1] := 5.15535E-01;
afSi[527, 0] := 6.35000E+03; afSi[527, 1] := 5.08167E-01;
afSi[528, 0] := 6.40000E+03; afSi[528, 1] := 5.00964E-01;
afSi[529, 0] := 6.45000E+03; afSi[529, 1] := 4.93915E-01;
afSi[530, 0] := 6.50000E+03; afSi[530, 1] := 4.87022E-01;
afSi[531, 0] := 6.55000E+03; afSi[531, 1] := 4.80279E-01;
afSi[532, 0] := 6.60000E+03; afSi[532, 1] := 4.73675E-01;
afSi[533, 0] := 6.65000E+03; afSi[533, 1] := 4.67207E-01;
afSi[534, 0] := 6.70000E+03; afSi[534, 1] := 4.60877E-01;
afSi[535, 0] := 6.75000E+03; afSi[535, 1] := 4.54682E-01;
afSi[536, 0] := 6.80000E+03; afSi[536, 1] := 4.48615E-01;
afSi[537, 0] := 6.85000E+03; afSi[537, 1] := 4.42675E-01;
afSi[538, 0] := 6.90000E+03; afSi[538, 1] := 4.36855E-01;
afSi[539, 0] := 6.95000E+03; afSi[539, 1] := 4.31151E-01;
afSi[540, 0] := 7.00000E+03; afSi[540, 1] := 4.25560E-01;
afSi[541, 0] := 7.05000E+03; afSi[541, 1] := 4.20081E-01;
afSi[542, 0] := 7.10000E+03; afSi[542, 1] := 4.14712E-01;
afSi[543, 0] := 7.15000E+03; afSi[543, 1] := 4.09450E-01;
afSi[544, 0] := 7.20000E+03; afSi[544, 1] := 4.04294E-01;
afSi[545, 0] := 7.25000E+03; afSi[545, 1] := 3.99235E-01;
afSi[546, 0] := 7.30000E+03; afSi[546, 1] := 3.94270E-01;
afSi[547, 0] := 7.35000E+03; afSi[547, 1] := 3.89406E-01;
afSi[548, 0] := 7.40000E+03; afSi[548, 1] := 3.84633E-01;
afSi[549, 0] := 7.45000E+03; afSi[549, 1] := 3.79947E-01;
afSi[550, 0] := 7.50000E+03; afSi[550, 1] := 3.75353E-01;
afSi[551, 0] := 7.55000E+03; afSi[551, 1] := 3.70843E-01;
afSi[552, 0] := 7.60000E+03; afSi[552, 1] := 3.66417E-01;
afSi[553, 0] := 7.65000E+03; afSi[553, 1] := 3.62071E-01;
afSi[554, 0] := 7.70000E+03; afSi[554, 1] := 3.57805E-01;
afSi[555, 0] := 7.75000E+03; afSi[555, 1] := 3.53618E-01;
afSi[556, 0] := 7.80000E+03; afSi[556, 1] := 3.49502E-01;
afSi[557, 0] := 7.85000E+03; afSi[557, 1] := 3.45461E-01;
afSi[558, 0] := 7.90000E+03; afSi[558, 1] := 3.41495E-01;
afSi[559, 0] := 7.95000E+03; afSi[559, 1] := 3.37563E-01;
afSi[560, 0] := 8.00000E+03; afSi[560, 1] := 3.33644E-01;
afSi[561, 0] := 8.05000E+03; afSi[561, 1] := 3.29688E-01;
afSi[562, 0] := 8.10000E+03; afSi[562, 1] := 3.25799E-01;
afSi[563, 0] := 8.15000E+03; afSi[563, 1] := 3.21979E-01;
afSi[564, 0] := 8.20000E+03; afSi[564, 1] := 3.18233E-01;
afSi[565, 0] := 8.25000E+03; afSi[565, 1] := 3.14552E-01;
afSi[566, 0] := 8.30000E+03; afSi[566, 1] := 3.10934E-01;
afSi[567, 0] := 8.35000E+03; afSi[567, 1] := 3.07377E-01;
afSi[568, 0] := 8.40000E+03; afSi[568, 1] := 3.03882E-01;
afSi[569, 0] := 8.45000E+03; afSi[569, 1] := 3.00446E-01;
afSi[570, 0] := 8.50000E+03; afSi[570, 1] := 2.97073E-01;
afSi[571, 0] := 8.55000E+03; afSi[571, 1] := 2.93760E-01;
afSi[572, 0] := 8.60000E+03; afSi[572, 1] := 2.90496E-01;
afSi[573, 0] := 8.65000E+03; afSi[573, 1] := 2.87286E-01;
afSi[574, 0] := 8.70000E+03; afSi[574, 1] := 2.84137E-01;
afSi[575, 0] := 8.75000E+03; afSi[575, 1] := 2.81038E-01;
afSi[576, 0] := 8.80000E+03; afSi[576, 1] := 2.77986E-01;
afSi[577, 0] := 8.85000E+03; afSi[577, 1] := 2.74976E-01;
afSi[578, 0] := 8.90000E+03; afSi[578, 1] := 2.72012E-01;
afSi[579, 0] := 8.95000E+03; afSi[579, 1] := 2.68954E-01;
afSi[580, 0] := 9.00000E+03; afSi[580, 1] := 2.65925E-01;
afSi[581, 0] := 9.05000E+03; afSi[581, 1] := 2.62952E-01;
afSi[582, 0] := 9.10000E+03; afSi[582, 1] := 2.60026E-01;
afSi[583, 0] := 9.15000E+03; afSi[583, 1] := 2.57142E-01;
afSi[584, 0] := 9.20000E+03; afSi[584, 1] := 2.54307E-01;
afSi[585, 0] := 9.25000E+03; afSi[585, 1] := 2.51519E-01;
afSi[586, 0] := 9.30000E+03; afSi[586, 1] := 2.48780E-01;
afSi[587, 0] := 9.35000E+03; afSi[587, 1] := 2.46086E-01;
afSi[588, 0] := 9.40000E+03; afSi[588, 1] := 2.43431E-01;
afSi[589, 0] := 9.45000E+03; afSi[589, 1] := 2.40817E-01;
afSi[590, 0] := 9.50000E+03; afSi[590, 1] := 2.38251E-01;
afSi[591, 0] := 9.55000E+03; afSi[591, 1] := 2.35726E-01;
afSi[592, 0] := 9.60000E+03; afSi[592, 1] := 2.33237E-01;
afSi[593, 0] := 9.65000E+03; afSi[593, 1] := 2.30787E-01;
afSi[594, 0] := 9.70000E+03; afSi[594, 1] := 2.28373E-01;
afSi[595, 0] := 9.75000E+03; afSi[595, 1] := 2.25998E-01;
afSi[596, 0] := 9.80000E+03; afSi[596, 1] := 2.23662E-01;
afSi[597, 0] := 9.85000E+03; afSi[597, 1] := 2.21361E-01;
afSi[598, 0] := 9.90000E+03; afSi[598, 1] := 2.19096E-01;
afSi[599, 0] := 9.95000E+03; afSi[599, 1] := 2.16865E-01;
afSi[600, 0] := 1.00000E+04; afSi[600, 1] := 2.14669E-01;
afSi[601, 0] := 1.00500E+04; afSi[601, 1] := 2.12504E-01;
afSi[602, 0] := 1.01000E+04; afSi[602, 1] := 2.10369E-01;
afSi[603, 0] := 1.01500E+04; afSi[603, 1] := 2.08267E-01;
afSi[604, 0] := 1.02000E+04; afSi[604, 1] := 2.06198E-01;
afSi[605, 0] := 1.02500E+04; afSi[605, 1] := 2.04159E-01;
afSi[606, 0] := 1.03000E+04; afSi[606, 1] := 2.02154E-01;
afSi[607, 0] := 1.03500E+04; afSi[607, 1] := 2.00176E-01;
afSi[608, 0] := 1.04000E+04; afSi[608, 1] := 1.98222E-01;
afSi[609, 0] := 1.04500E+04; afSi[609, 1] := 1.96297E-01;
afSi[610, 0] := 1.05000E+04; afSi[610, 1] := 1.94404E-01;
afSi[611, 0] := 1.05500E+04; afSi[611, 1] := 1.92538E-01;
afSi[612, 0] := 1.06000E+04; afSi[612, 1] := 1.90695E-01;
afSi[613, 0] := 1.06500E+04; afSi[613, 1] := 1.88878E-01;
afSi[614, 0] := 1.07000E+04; afSi[614, 1] := 1.87092E-01;
afSi[615, 0] := 1.07500E+04; afSi[615, 1] := 1.85331E-01;
afSi[616, 0] := 1.08000E+04; afSi[616, 1] := 1.83594E-01;
afSi[617, 0] := 1.08500E+04; afSi[617, 1] := 1.81879E-01;
afSi[618, 0] := 1.09000E+04; afSi[618, 1] := 1.80188E-01;
afSi[619, 0] := 1.09500E+04; afSi[619, 1] := 1.78519E-01;
afSi[620, 0] := 1.10000E+04; afSi[620, 1] := 1.76873E-01;
afSi[621, 0] := 1.10500E+04; afSi[621, 1] := 1.75248E-01;
afSi[622, 0] := 1.11000E+04; afSi[622, 1] := 1.73647E-01;
afSi[623, 0] := 1.11500E+04; afSi[623, 1] := 1.72070E-01;
afSi[624, 0] := 1.12000E+04; afSi[624, 1] := 1.70515E-01;
afSi[625, 0] := 1.12500E+04; afSi[625, 1] := 1.68980E-01;
afSi[626, 0] := 1.13000E+04; afSi[626, 1] := 1.67466E-01;
afSi[627, 0] := 1.13500E+04; afSi[627, 1] := 1.65970E-01;
afSi[628, 0] := 1.14000E+04; afSi[628, 1] := 1.64492E-01;
afSi[629, 0] := 1.14500E+04; afSi[629, 1] := 1.63035E-01;
afSi[630, 0] := 1.15000E+04; afSi[630, 1] := 1.61598E-01;
afSi[631, 0] := 1.15500E+04; afSi[631, 1] := 1.60179E-01;
afSi[632, 0] := 1.16000E+04; afSi[632, 1] := 1.58781E-01;
afSi[633, 0] := 1.16500E+04; afSi[633, 1] := 1.57401E-01;
afSi[634, 0] := 1.17000E+04; afSi[634, 1] := 1.56037E-01;
afSi[635, 0] := 1.17500E+04; afSi[635, 1] := 1.54690E-01;
afSi[636, 0] := 1.18000E+04; afSi[636, 1] := 1.53363E-01;
afSi[637, 0] := 1.18500E+04; afSi[637, 1] := 1.52054E-01;
afSi[638, 0] := 1.19000E+04; afSi[638, 1] := 1.50760E-01;
afSi[639, 0] := 1.19500E+04; afSi[639, 1] := 1.49478E-01;
afSi[640, 0] := 1.20000E+04; afSi[640, 1] := 1.48213E-01;
afSi[641, 0] := 1.20500E+04; afSi[641, 1] := 1.46967E-01;
afSi[642, 0] := 1.21000E+04; afSi[642, 1] := 1.45738E-01;
afSi[643, 0] := 1.21500E+04; afSi[643, 1] := 1.44523E-01;
afSi[644, 0] := 1.22000E+04; afSi[644, 1] := 1.43324E-01;
afSi[645, 0] := 1.22500E+04; afSi[645, 1] := 1.42140E-01;
afSi[646, 0] := 1.23000E+04; afSi[646, 1] := 1.40967E-01;
afSi[647, 0] := 1.23500E+04; afSi[647, 1] := 1.39808E-01;
afSi[648, 0] := 1.24000E+04; afSi[648, 1] := 1.38664E-01;
afSi[649, 0] := 1.24500E+04; afSi[649, 1] := 1.37535E-01;
afSi[650, 0] := 1.25000E+04; afSi[650, 1] := 1.36420E-01;
afSi[651, 0] := 1.25500E+04; afSi[651, 1] := 1.35319E-01;
afSi[652, 0] := 1.26000E+04; afSi[652, 1] := 1.34232E-01;
afSi[653, 0] := 1.26500E+04; afSi[653, 1] := 1.33156E-01;
afSi[654, 0] := 1.27000E+04; afSi[654, 1] := 1.32093E-01;
afSi[655, 0] := 1.27500E+04; afSi[655, 1] := 1.31042E-01;
afSi[656, 0] := 1.28000E+04; afSi[656, 1] := 1.30006E-01;
afSi[657, 0] := 1.28500E+04; afSi[657, 1] := 1.28983E-01;
afSi[658, 0] := 1.29000E+04; afSi[658, 1] := 1.27970E-01;
afSi[659, 0] := 1.29500E+04; afSi[659, 1] := 1.26970E-01;
afSi[660, 0] := 1.30000E+04; afSi[660, 1] := 1.25980E-01;
afSi[661, 0] := 1.30500E+04; afSi[661, 1] := 1.25002E-01;
afSi[662, 0] := 1.31000E+04; afSi[662, 1] := 1.24035E-01;
afSi[663, 0] := 1.31500E+04; afSi[663, 1] := 1.23079E-01;
afSi[664, 0] := 1.32000E+04; afSi[664, 1] := 1.22134E-01;
afSi[665, 0] := 1.32500E+04; afSi[665, 1] := 1.21200E-01;
afSi[666, 0] := 1.33000E+04; afSi[666, 1] := 1.20277E-01;
afSi[667, 0] := 1.33500E+04; afSi[667, 1] := 1.19364E-01;
afSi[668, 0] := 1.34000E+04; afSi[668, 1] := 1.18461E-01;
afSi[669, 0] := 1.34500E+04; afSi[669, 1] := 1.17569E-01;
afSi[670, 0] := 1.35000E+04; afSi[670, 1] := 1.16687E-01;
afSi[671, 0] := 1.35500E+04; afSi[671, 1] := 1.15814E-01;
afSi[672, 0] := 1.36000E+04; afSi[672, 1] := 1.14949E-01;
afSi[673, 0] := 1.36500E+04; afSi[673, 1] := 1.14093E-01;
afSi[674, 0] := 1.37000E+04; afSi[674, 1] := 1.13251E-01;
afSi[675, 0] := 1.37500E+04; afSi[675, 1] := 1.12419E-01;
afSi[676, 0] := 1.38000E+04; afSi[676, 1] := 1.11596E-01;
afSi[677, 0] := 1.38500E+04; afSi[677, 1] := 1.10777E-01;
afSi[678, 0] := 1.39000E+04; afSi[678, 1] := 1.09967E-01;
afSi[679, 0] := 1.39500E+04; afSi[679, 1] := 1.09166E-01;
afSi[680, 0] := 1.40000E+04; afSi[680, 1] := 1.08379E-01;
afSi[681, 0] := 1.40500E+04; afSi[681, 1] := 1.07600E-01;
afSi[682, 0] := 1.41000E+04; afSi[682, 1] := 1.06827E-01;
afSi[683, 0] := 1.41500E+04; afSi[683, 1] := 1.06059E-01;
afSi[684, 0] := 1.42000E+04; afSi[684, 1] := 1.05300E-01;
afSi[685, 0] := 1.42500E+04; afSi[685, 1] := 1.04551E-01;
afSi[686, 0] := 1.43000E+04; afSi[686, 1] := 1.03810E-01;
afSi[687, 0] := 1.43500E+04; afSi[687, 1] := 1.03077E-01;
afSi[688, 0] := 1.44000E+04; afSi[688, 1] := 1.02351E-01;
afSi[689, 0] := 1.44500E+04; afSi[689, 1] := 1.01633E-01;
afSi[690, 0] := 1.45000E+04; afSi[690, 1] := 1.00922E-01;
afSi[691, 0] := 1.45500E+04; afSi[691, 1] := 1.00221E-01;
afSi[692, 0] := 1.46000E+04; afSi[692, 1] := 9.95261E-02;
afSi[693, 0] := 1.46500E+04; afSi[693, 1] := 9.88388E-02;
afSi[694, 0] := 1.47000E+04; afSi[694, 1] := 9.81578E-02;
afSi[695, 0] := 1.47500E+04; afSi[695, 1] := 9.74838E-02;
afSi[696, 0] := 1.48000E+04; afSi[696, 1] := 9.68166E-02;
afSi[697, 0] := 1.48500E+04; afSi[697, 1] := 9.61558E-02;
afSi[698, 0] := 1.49000E+04; afSi[698, 1] := 9.55016E-02;
afSi[699, 0] := 1.49500E+04; afSi[699, 1] := 9.48542E-02;
afSi[700, 0] := 1.50000E+04; afSi[700, 1] := 9.42136E-02;
afSi[701, 0] := 1.50500E+04; afSi[701, 1] := 9.35795E-02;
afSi[702, 0] := 1.51000E+04; afSi[702, 1] := 9.29516E-02;
afSi[703, 0] := 1.51500E+04; afSi[703, 1] := 9.23298E-02;
afSi[704, 0] := 1.52000E+04; afSi[704, 1] := 9.17141E-02;
afSi[705, 0] := 1.52500E+04; afSi[705, 1] := 9.11046E-02;
afSi[706, 0] := 1.53000E+04; afSi[706, 1] := 9.05014E-02;
afSi[707, 0] := 1.53500E+04; afSi[707, 1] := 8.99041E-02;
afSi[708, 0] := 1.54000E+04; afSi[708, 1] := 8.93126E-02;
afSi[709, 0] := 1.54500E+04; afSi[709, 1] := 8.87268E-02;
afSi[710, 0] := 1.55000E+04; afSi[710, 1] := 8.81467E-02;
afSi[711, 0] := 1.55500E+04; afSi[711, 1] := 8.75723E-02;
afSi[712, 0] := 1.56000E+04; afSi[712, 1] := 8.70035E-02;
afSi[713, 0] := 1.56500E+04; afSi[713, 1] := 8.64402E-02;
afSi[714, 0] := 1.57000E+04; afSi[714, 1] := 8.58823E-02;
afSi[715, 0] := 1.57500E+04; afSi[715, 1] := 8.53298E-02;
afSi[716, 0] := 1.58000E+04; afSi[716, 1] := 8.47826E-02;
afSi[717, 0] := 1.58500E+04; afSi[717, 1] := 8.42406E-02;
afSi[718, 0] := 1.59000E+04; afSi[718, 1] := 8.37037E-02;
afSi[719, 0] := 1.59500E+04; afSi[719, 1] := 8.31718E-02;
afSi[720, 0] := 1.60000E+04; afSi[720, 1] := 8.26450E-02;
afSi[721, 0] := 1.60500E+04; afSi[721, 1] := 8.21232E-02;
afSi[722, 0] := 1.61000E+04; afSi[722, 1] := 8.16063E-02;
afSi[723, 0] := 1.61500E+04; afSi[723, 1] := 8.10943E-02;
afSi[724, 0] := 1.62000E+04; afSi[724, 1] := 8.05871E-02;
afSi[725, 0] := 1.62500E+04; afSi[725, 1] := 8.00846E-02;
afSi[726, 0] := 1.63000E+04; afSi[726, 1] := 7.95868E-02;
afSi[727, 0] := 1.63500E+04; afSi[727, 1] := 7.90936E-02;
afSi[728, 0] := 1.64000E+04; afSi[728, 1] := 7.86052E-02;
afSi[729, 0] := 1.64500E+04; afSi[729, 1] := 7.81212E-02;
afSi[730, 0] := 1.65000E+04; afSi[730, 1] := 7.76417E-02;
afSi[731, 0] := 1.65500E+04; afSi[731, 1] := 7.71664E-02;
afSi[732, 0] := 1.66000E+04; afSi[732, 1] := 7.66954E-02;
afSi[733, 0] := 1.66500E+04; afSi[733, 1] := 7.62286E-02;
afSi[734, 0] := 1.67000E+04; afSi[734, 1] := 7.57661E-02;
afSi[735, 0] := 1.67500E+04; afSi[735, 1] := 7.53078E-02;
afSi[736, 0] := 1.68000E+04; afSi[736, 1] := 7.48536E-02;
afSi[737, 0] := 1.68500E+04; afSi[737, 1] := 7.44035E-02;
afSi[738, 0] := 1.69000E+04; afSi[738, 1] := 7.39573E-02;
afSi[739, 0] := 1.69500E+04; afSi[739, 1] := 7.35150E-02;
afSi[740, 0] := 1.70000E+04; afSi[740, 1] := 7.30767E-02;
afSi[741, 0] := 1.70500E+04; afSi[741, 1] := 7.26424E-02;
afSi[742, 0] := 1.71000E+04; afSi[742, 1] := 7.22119E-02;
afSi[743, 0] := 1.71500E+04; afSi[743, 1] := 7.17852E-02;
afSi[744, 0] := 1.72000E+04; afSi[744, 1] := 7.13623E-02;
afSi[745, 0] := 1.72500E+04; afSi[745, 1] := 7.09433E-02;
afSi[746, 0] := 1.73000E+04; afSi[746, 1] := 7.05280E-02;
afSi[747, 0] := 1.73500E+04; afSi[747, 1] := 7.01163E-02;
afSi[748, 0] := 1.74000E+04; afSi[748, 1] := 6.97080E-02;
afSi[749, 0] := 1.74500E+04; afSi[749, 1] := 6.93032E-02;
afSi[750, 0] := 1.75000E+04; afSi[750, 1] := 6.89019E-02;
afSi[751, 0] := 1.75500E+04; afSi[751, 1] := 6.85041E-02;
afSi[752, 0] := 1.76000E+04; afSi[752, 1] := 6.81097E-02;
afSi[753, 0] := 1.76500E+04; afSi[753, 1] := 6.77186E-02;
afSi[754, 0] := 1.77000E+04; afSi[754, 1] := 6.73310E-02;
afSi[755, 0] := 1.77500E+04; afSi[755, 1] := 6.69467E-02;
afSi[756, 0] := 1.78000E+04; afSi[756, 1] := 6.65658E-02;
afSi[757, 0] := 1.78500E+04; afSi[757, 1] := 6.61880E-02;
afSi[758, 0] := 1.79000E+04; afSi[758, 1] := 6.58134E-02;
afSi[759, 0] := 1.79500E+04; afSi[759, 1] := 6.54417E-02;
afSi[760, 0] := 1.80000E+04; afSi[760, 1] := 6.50732E-02;
afSi[761, 0] := 1.80500E+04; afSi[761, 1] := 6.47078E-02;
afSi[762, 0] := 1.81000E+04; afSi[762, 1] := 6.43455E-02;
afSi[763, 0] := 1.81500E+04; afSi[763, 1] := 6.39864E-02;
afSi[764, 0] := 1.82000E+04; afSi[764, 1] := 6.36301E-02;
afSi[765, 0] := 1.82500E+04; afSi[765, 1] := 6.32769E-02;
afSi[766, 0] := 1.83000E+04; afSi[766, 1] := 6.29266E-02;
afSi[767, 0] := 1.83500E+04; afSi[767, 1] := 6.25792E-02;
afSi[768, 0] := 1.84000E+04; afSi[768, 1] := 6.22347E-02;
afSi[769, 0] := 1.84500E+04; afSi[769, 1] := 6.18929E-02;
afSi[770, 0] := 1.85000E+04; afSi[770, 1] := 6.15539E-02;
afSi[771, 0] := 1.85500E+04; afSi[771, 1] := 6.12176E-02;
afSi[772, 0] := 1.86000E+04; afSi[772, 1] := 6.08841E-02;
afSi[773, 0] := 1.86500E+04; afSi[773, 1] := 6.05533E-02;
afSi[774, 0] := 1.87000E+04; afSi[774, 1] := 6.02252E-02;
afSi[775, 0] := 1.87500E+04; afSi[775, 1] := 5.98998E-02;
afSi[776, 0] := 1.88000E+04; afSi[776, 1] := 5.95770E-02;
afSi[777, 0] := 1.88500E+04; afSi[777, 1] := 5.92570E-02;
afSi[778, 0] := 1.89000E+04; afSi[778, 1] := 5.89395E-02;
afSi[779, 0] := 1.89500E+04; afSi[779, 1] := 5.86245E-02;
afSi[780, 0] := 1.90000E+04; afSi[780, 1] := 5.83119E-02;
afSi[781, 0] := 1.90500E+04; afSi[781, 1] := 5.80017E-02;
afSi[782, 0] := 1.91000E+04; afSi[782, 1] := 5.76940E-02;
afSi[783, 0] := 1.91500E+04; afSi[783, 1] := 5.73887E-02;
afSi[784, 0] := 1.92000E+04; afSi[784, 1] := 5.70857E-02;
afSi[785, 0] := 1.92500E+04; afSi[785, 1] := 5.67851E-02;
afSi[786, 0] := 1.93000E+04; afSi[786, 1] := 5.64869E-02;
afSi[787, 0] := 1.93500E+04; afSi[787, 1] := 5.61909E-02;
afSi[788, 0] := 1.94000E+04; afSi[788, 1] := 5.58976E-02;
afSi[789, 0] := 1.94500E+04; afSi[789, 1] := 5.56065E-02;
afSi[790, 0] := 1.95000E+04; afSi[790, 1] := 5.53177E-02;
afSi[791, 0] := 1.95500E+04; afSi[791, 1] := 5.50312E-02;
afSi[792, 0] := 1.96000E+04; afSi[792, 1] := 5.47467E-02;
afSi[793, 0] := 1.96500E+04; afSi[793, 1] := 5.44644E-02;
afSi[794, 0] := 1.97000E+04; afSi[794, 1] := 5.41843E-02;
afSi[795, 0] := 1.97500E+04; afSi[795, 1] := 5.39064E-02;
afSi[796, 0] := 1.98000E+04; afSi[796, 1] := 5.36305E-02;
afSi[797, 0] := 1.98500E+04; afSi[797, 1] := 5.33568E-02;
afSi[798, 0] := 1.99000E+04; afSi[798, 1] := 5.30851E-02;
afSi[799, 0] := 1.99500E+04; afSi[799, 1] := 5.28155E-02;
afSi[800, 0] := 2.00000E+04; afSi[800, 1] := 5.25478E-02;
afSi[801, 0] := 2.00500E+04; afSi[801, 1] := 5.22822E-02;
afSi[802, 0] := 2.01000E+04; afSi[802, 1] := 5.20185E-02;
afSi[803, 0] := 2.01500E+04; afSi[803, 1] := 5.17569E-02;
afSi[804, 0] := 2.02000E+04; afSi[804, 1] := 5.14973E-02;
afSi[805, 0] := 2.02500E+04; afSi[805, 1] := 5.12398E-02;
afSi[806, 0] := 2.03000E+04; afSi[806, 1] := 5.09841E-02;
afSi[807, 0] := 2.03500E+04; afSi[807, 1] := 5.07304E-02;
afSi[808, 0] := 2.04000E+04; afSi[808, 1] := 5.04786E-02;
afSi[809, 0] := 2.04500E+04; afSi[809, 1] := 5.02286E-02;
afSi[810, 0] := 2.05000E+04; afSi[810, 1] := 4.99806E-02;
afSi[811, 0] := 2.05500E+04; afSi[811, 1] := 4.97343E-02;
afSi[812, 0] := 2.06000E+04; afSi[812, 1] := 4.94895E-02;
afSi[813, 0] := 2.06500E+04; afSi[813, 1] := 4.92465E-02;
afSi[814, 0] := 2.07000E+04; afSi[814, 1] := 4.90053E-02;
afSi[815, 0] := 2.07500E+04; afSi[815, 1] := 4.87659E-02;
afSi[816, 0] := 2.08000E+04; afSi[816, 1] := 4.85285E-02;
afSi[817, 0] := 2.08500E+04; afSi[817, 1] := 4.82928E-02;
afSi[818, 0] := 2.09000E+04; afSi[818, 1] := 4.80588E-02;
afSi[819, 0] := 2.09500E+04; afSi[819, 1] := 4.78264E-02;
afSi[820, 0] := 2.10000E+04; afSi[820, 1] := 4.75957E-02;
afSi[821, 0] := 2.10500E+04; afSi[821, 1] := 4.73666E-02;
afSi[822, 0] := 2.11000E+04; afSi[822, 1] := 4.71392E-02;
afSi[823, 0] := 2.11500E+04; afSi[823, 1] := 4.69134E-02;
afSi[824, 0] := 2.12000E+04; afSi[824, 1] := 4.66891E-02;
afSi[825, 0] := 2.12500E+04; afSi[825, 1] := 4.64665E-02;
afSi[826, 0] := 2.13000E+04; afSi[826, 1] := 4.62454E-02;
afSi[827, 0] := 2.13500E+04; afSi[827, 1] := 4.60260E-02;
afSi[828, 0] := 2.14000E+04; afSi[828, 1] := 4.58081E-02;
afSi[829, 0] := 2.14500E+04; afSi[829, 1] := 4.55917E-02;
afSi[830, 0] := 2.15000E+04; afSi[830, 1] := 4.53769E-02;
afSi[831, 0] := 2.15500E+04; afSi[831, 1] := 4.51636E-02;
afSi[832, 0] := 2.16000E+04; afSi[832, 1] := 4.49518E-02;
afSi[833, 0] := 2.16500E+04; afSi[833, 1] := 4.47414E-02;
afSi[834, 0] := 2.17000E+04; afSi[834, 1] := 4.45325E-02;
afSi[835, 0] := 2.17500E+04; afSi[835, 1] := 4.43250E-02;
afSi[836, 0] := 2.18000E+04; afSi[836, 1] := 4.41189E-02;
afSi[837, 0] := 2.18500E+04; afSi[837, 1] := 4.39143E-02;
afSi[838, 0] := 2.19000E+04; afSi[838, 1] := 4.37111E-02;
afSi[839, 0] := 2.19500E+04; afSi[839, 1] := 4.35093E-02;
afSi[840, 0] := 2.20000E+04; afSi[840, 1] := 4.33089E-02;
afSi[841, 0] := 2.20500E+04; afSi[841, 1] := 4.31099E-02;
afSi[842, 0] := 2.21000E+04; afSi[842, 1] := 4.29124E-02;
afSi[843, 0] := 2.21500E+04; afSi[843, 1] := 4.27161E-02;
afSi[844, 0] := 2.22000E+04; afSi[844, 1] := 4.25212E-02;
afSi[845, 0] := 2.22500E+04; afSi[845, 1] := 4.23277E-02;
afSi[846, 0] := 2.23000E+04; afSi[846, 1] := 4.21353E-02;
afSi[847, 0] := 2.23500E+04; afSi[847, 1] := 4.19443E-02;
afSi[848, 0] := 2.24000E+04; afSi[848, 1] := 4.17546E-02;
afSi[849, 0] := 2.24500E+04; afSi[849, 1] := 4.15662E-02;
afSi[850, 0] := 2.25000E+04; afSi[850, 1] := 4.13790E-02;
afSi[851, 0] := 2.25500E+04; afSi[851, 1] := 4.11931E-02;
afSi[852, 0] := 2.26000E+04; afSi[852, 1] := 4.10084E-02;
afSi[853, 0] := 2.26500E+04; afSi[853, 1] := 4.08250E-02;
afSi[854, 0] := 2.27000E+04; afSi[854, 1] := 4.06428E-02;
afSi[855, 0] := 2.27500E+04; afSi[855, 1] := 4.04619E-02;
afSi[856, 0] := 2.28000E+04; afSi[856, 1] := 4.02822E-02;
afSi[857, 0] := 2.28500E+04; afSi[857, 1] := 4.01037E-02;
afSi[858, 0] := 2.29000E+04; afSi[858, 1] := 3.99264E-02;
afSi[859, 0] := 2.29500E+04; afSi[859, 1] := 3.97502E-02;
afSi[860, 0] := 2.30000E+04; afSi[860, 1] := 3.95752E-02;
afSi[861, 0] := 2.30500E+04; afSi[861, 1] := 3.94013E-02;
afSi[862, 0] := 2.31000E+04; afSi[862, 1] := 3.92285E-02;
afSi[863, 0] := 2.31500E+04; afSi[863, 1] := 3.90569E-02;
afSi[864, 0] := 2.32000E+04; afSi[864, 1] := 3.88862E-02;
afSi[865, 0] := 2.32500E+04; afSi[865, 1] := 3.87166E-02;
afSi[866, 0] := 2.33000E+04; afSi[866, 1] := 3.85481E-02;
afSi[867, 0] := 2.33500E+04; afSi[867, 1] := 3.83807E-02;
afSi[868, 0] := 2.34000E+04; afSi[868, 1] := 3.82145E-02;
afSi[869, 0] := 2.34500E+04; afSi[869, 1] := 3.80495E-02;
afSi[870, 0] := 2.35000E+04; afSi[870, 1] := 3.78856E-02;
afSi[871, 0] := 2.35500E+04; afSi[871, 1] := 3.77228E-02;
afSi[872, 0] := 2.36000E+04; afSi[872, 1] := 3.75610E-02;
afSi[873, 0] := 2.36500E+04; afSi[873, 1] := 3.74001E-02;
afSi[874, 0] := 2.37000E+04; afSi[874, 1] := 3.72401E-02;
afSi[875, 0] := 2.37500E+04; afSi[875, 1] := 3.70811E-02;
afSi[876, 0] := 2.38000E+04; afSi[876, 1] := 3.69231E-02;
afSi[877, 0] := 2.38500E+04; afSi[877, 1] := 3.67662E-02;
afSi[878, 0] := 2.39000E+04; afSi[878, 1] := 3.66104E-02;
afSi[879, 0] := 2.39500E+04; afSi[879, 1] := 3.64556E-02;
afSi[880, 0] := 2.40000E+04; afSi[880, 1] := 3.63018E-02;
afSi[881, 0] := 2.40500E+04; afSi[881, 1] := 3.61490E-02;
afSi[882, 0] := 2.41000E+04; afSi[882, 1] := 3.59971E-02;
afSi[883, 0] := 2.41500E+04; afSi[883, 1] := 3.58460E-02;
afSi[884, 0] := 2.42000E+04; afSi[884, 1] := 3.56959E-02;
afSi[885, 0] := 2.42500E+04; afSi[885, 1] := 3.55467E-02;
afSi[886, 0] := 2.43000E+04; afSi[886, 1] := 3.53985E-02;
afSi[887, 0] := 2.43500E+04; afSi[887, 1] := 3.52512E-02;
afSi[888, 0] := 2.44000E+04; afSi[888, 1] := 3.51049E-02;
afSi[889, 0] := 2.44500E+04; afSi[889, 1] := 3.49595E-02;
afSi[890, 0] := 2.45000E+04; afSi[890, 1] := 3.48150E-02;
afSi[891, 0] := 2.45500E+04; afSi[891, 1] := 3.46714E-02;
afSi[892, 0] := 2.46000E+04; afSi[892, 1] := 3.45287E-02;
afSi[893, 0] := 2.46500E+04; afSi[893, 1] := 3.43868E-02;
afSi[894, 0] := 2.47000E+04; afSi[894, 1] := 3.42458E-02;
afSi[895, 0] := 2.47500E+04; afSi[895, 1] := 3.41057E-02;
afSi[896, 0] := 2.48000E+04; afSi[896, 1] := 3.39664E-02;
afSi[897, 0] := 2.48500E+04; afSi[897, 1] := 3.38279E-02;
afSi[898, 0] := 2.49000E+04; afSi[898, 1] := 3.36901E-02;
afSi[899, 0] := 2.49500E+04; afSi[899, 1] := 3.35532E-02;
afSi[900, 0] := 2.50000E+04; afSi[900, 1] := 3.34171E-02;
afSi[901, 0] := 2.50500E+04; afSi[901, 1] := 3.32819E-02;
afSi[902, 0] := 2.51000E+04; afSi[902, 1] := 3.31475E-02;
afSi[903, 0] := 2.51500E+04; afSi[903, 1] := 3.30139E-02;
afSi[904, 0] := 2.52000E+04; afSi[904, 1] := 3.28812E-02;
afSi[905, 0] := 2.52500E+04; afSi[905, 1] := 3.27492E-02;
afSi[906, 0] := 2.53000E+04; afSi[906, 1] := 3.26181E-02;
afSi[907, 0] := 2.53500E+04; afSi[907, 1] := 3.24878E-02;
afSi[908, 0] := 2.54000E+04; afSi[908, 1] := 3.23583E-02;
afSi[909, 0] := 2.54500E+04; afSi[909, 1] := 3.22296E-02;
afSi[910, 0] := 2.55000E+04; afSi[910, 1] := 3.21017E-02;
afSi[911, 0] := 2.55500E+04; afSi[911, 1] := 3.19745E-02;
afSi[912, 0] := 2.56000E+04; afSi[912, 1] := 3.18480E-02;
afSi[913, 0] := 2.56500E+04; afSi[913, 1] := 3.17222E-02;
afSi[914, 0] := 2.57000E+04; afSi[914, 1] := 3.15970E-02;
afSi[915, 0] := 2.57500E+04; afSi[915, 1] := 3.14726E-02;
afSi[916, 0] := 2.58000E+04; afSi[916, 1] := 3.13490E-02;
afSi[917, 0] := 2.58500E+04; afSi[917, 1] := 3.12261E-02;
afSi[918, 0] := 2.59000E+04; afSi[918, 1] := 3.11039E-02;
afSi[919, 0] := 2.59500E+04; afSi[919, 1] := 3.09824E-02;
afSi[920, 0] := 2.60000E+04; afSi[920, 1] := 3.08617E-02;
afSi[921, 0] := 2.60500E+04; afSi[921, 1] := 3.07416E-02;
afSi[922, 0] := 2.61000E+04; afSi[922, 1] := 3.06223E-02;
afSi[923, 0] := 2.61500E+04; afSi[923, 1] := 3.05037E-02;
afSi[924, 0] := 2.62000E+04; afSi[924, 1] := 3.03859E-02;
afSi[925, 0] := 2.62500E+04; afSi[925, 1] := 3.02687E-02;
afSi[926, 0] := 2.63000E+04; afSi[926, 1] := 3.01521E-02;
afSi[927, 0] := 2.63500E+04; afSi[927, 1] := 3.00363E-02;
afSi[928, 0] := 2.64000E+04; afSi[928, 1] := 2.99210E-02;
afSi[929, 0] := 2.64500E+04; afSi[929, 1] := 2.98065E-02;
afSi[930, 0] := 2.65000E+04; afSi[930, 1] := 2.96925E-02;
afSi[931, 0] := 2.65500E+04; afSi[931, 1] := 2.95793E-02;
afSi[932, 0] := 2.66000E+04; afSi[932, 1] := 2.94666E-02;
afSi[933, 0] := 2.66500E+04; afSi[933, 1] := 2.93519E-02;
afSi[934, 0] := 2.67000E+04; afSi[934, 1] := 2.92369E-02;
afSi[935, 0] := 2.67500E+04; afSi[935, 1] := 2.91226E-02;
afSi[936, 0] := 2.68000E+04; afSi[936, 1] := 2.90090E-02;
afSi[937, 0] := 2.68500E+04; afSi[937, 1] := 2.88960E-02;
afSi[938, 0] := 2.69000E+04; afSi[938, 1] := 2.87828E-02;
afSi[939, 0] := 2.69500E+04; afSi[939, 1] := 2.86691E-02;
afSi[940, 0] := 2.70000E+04; afSi[940, 1] := 2.85560E-02;
afSi[941, 0] := 2.70500E+04; afSi[941, 1] := 2.84437E-02;
afSi[942, 0] := 2.71000E+04; afSi[942, 1] := 2.83319E-02;
afSi[943, 0] := 2.71500E+04; afSi[943, 1] := 2.82208E-02;
afSi[944, 0] := 2.72000E+04; afSi[944, 1] := 2.81106E-02;
afSi[945, 0] := 2.72500E+04; afSi[945, 1] := 2.80011E-02;
afSi[946, 0] := 2.73000E+04; afSi[946, 1] := 2.78921E-02;
afSi[947, 0] := 2.73500E+04; afSi[947, 1] := 2.77838E-02;
afSi[948, 0] := 2.74000E+04; afSi[948, 1] := 2.76761E-02;
afSi[949, 0] := 2.74500E+04; afSi[949, 1] := 2.75690E-02;
afSi[950, 0] := 2.75000E+04; afSi[950, 1] := 2.74624E-02;
afSi[951, 0] := 2.75500E+04; afSi[951, 1] := 2.73565E-02;
afSi[952, 0] := 2.76000E+04; afSi[952, 1] := 2.72511E-02;
afSi[953, 0] := 2.76500E+04; afSi[953, 1] := 2.71464E-02;
afSi[954, 0] := 2.77000E+04; afSi[954, 1] := 2.70422E-02;
afSi[955, 0] := 2.77500E+04; afSi[955, 1] := 2.69386E-02;
afSi[956, 0] := 2.78000E+04; afSi[956, 1] := 2.68356E-02;
afSi[957, 0] := 2.78500E+04; afSi[957, 1] := 2.67331E-02;
afSi[958, 0] := 2.79000E+04; afSi[958, 1] := 2.66313E-02;
afSi[959, 0] := 2.79500E+04; afSi[959, 1] := 2.65300E-02;
afSi[960, 0] := 2.80000E+04; afSi[960, 1] := 2.64292E-02;
afSi[961, 0] := 2.80500E+04; afSi[961, 1] := 2.63291E-02;
afSi[962, 0] := 2.81000E+04; afSi[962, 1] := 2.62295E-02;
afSi[963, 0] := 2.81500E+04; afSi[963, 1] := 2.61305E-02;
afSi[964, 0] := 2.82000E+04; afSi[964, 1] := 2.60320E-02;
afSi[965, 0] := 2.82500E+04; afSi[965, 1] := 2.59340E-02;
afSi[966, 0] := 2.83000E+04; afSi[966, 1] := 2.58365E-02;
afSi[967, 0] := 2.83500E+04; afSi[967, 1] := 2.57395E-02;
afSi[968, 0] := 2.84000E+04; afSi[968, 1] := 2.56431E-02;
afSi[969, 0] := 2.84500E+04; afSi[969, 1] := 2.55472E-02;
afSi[970, 0] := 2.85000E+04; afSi[970, 1] := 2.54518E-02;
afSi[971, 0] := 2.85500E+04; afSi[971, 1] := 2.53569E-02;
afSi[972, 0] := 2.86000E+04; afSi[972, 1] := 2.52627E-02;
afSi[973, 0] := 2.86500E+04; afSi[973, 1] := 2.51690E-02;
afSi[974, 0] := 2.87000E+04; afSi[974, 1] := 2.50757E-02;
afSi[975, 0] := 2.87500E+04; afSi[975, 1] := 2.49830E-02;
afSi[976, 0] := 2.88000E+04; afSi[976, 1] := 2.48908E-02;
afSi[977, 0] := 2.88500E+04; afSi[977, 1] := 2.47991E-02;
afSi[978, 0] := 2.89000E+04; afSi[978, 1] := 2.47078E-02;
afSi[979, 0] := 2.89500E+04; afSi[979, 1] := 2.46171E-02;
afSi[980, 0] := 2.90000E+04; afSi[980, 1] := 2.45268E-02;
afSi[981, 0] := 2.90500E+04; afSi[981, 1] := 2.44371E-02;
afSi[982, 0] := 2.91000E+04; afSi[982, 1] := 2.43478E-02;
afSi[983, 0] := 2.91500E+04; afSi[983, 1] := 2.42590E-02;
afSi[984, 0] := 2.92000E+04; afSi[984, 1] := 2.41706E-02;
afSi[985, 0] := 2.92500E+04; afSi[985, 1] := 2.40828E-02;
afSi[986, 0] := 2.93000E+04; afSi[986, 1] := 2.39954E-02;
afSi[987, 0] := 2.93500E+04; afSi[987, 1] := 2.39085E-02;
afSi[988, 0] := 2.94000E+04; afSi[988, 1] := 2.38220E-02;
afSi[989, 0] := 2.94500E+04; afSi[989, 1] := 2.37361E-02;
afSi[990, 0] := 2.95000E+04; afSi[990, 1] := 2.36506E-02;
afSi[991, 0] := 2.95500E+04; afSi[991, 1] := 2.35656E-02;
afSi[992, 0] := 2.96000E+04; afSi[992, 1] := 2.34810E-02;
afSi[993, 0] := 2.96500E+04; afSi[993, 1] := 2.33968E-02;
afSi[994, 0] := 2.97000E+04; afSi[994, 1] := 2.33131E-02;
afSi[995, 0] := 2.97500E+04; afSi[995, 1] := 2.32298E-02;
afSi[996, 0] := 2.98000E+04; afSi[996, 1] := 2.31469E-02;
afSi[997, 0] := 2.98500E+04; afSi[997, 1] := 2.30644E-02;
afSi[998, 0] := 2.99000E+04; afSi[998, 1] := 2.29824E-02;
afSi[999, 0] := 2.99500E+04; afSi[999, 1] := 2.29008E-02;
END_METHOD

END_FUNCTION_BLOCK

(* stored: Version 1.1.0.1
   POU FB_f2Chantler: Id {758ca0c8-4f2b-4733-8a38-5b55dddc9fe1}, SpecialFunc None
   Method GetMissingLookupTableForElementMsg: Id {34404fc1-6e1d-40e0-9a7a-7ca0105727ac}
   Method GetPhotonEnergyOutOfTableRangeMsg: Id {7cedaa09-f02a-492a-81e2-8d44d5becbf7}
   Method MakeTables: Id {d3bdfca8-f75b-4e24-9f6b-61aa9de92a99} *)
